{attribute 'GeneratedUsingTerminal: EJ3214-0000-0016'}
{attribute addProperty BoxType "EJ3214-0000-0016"}
{attribute addProperty Id "StatusAT %I*Status_68C33E995ValueAT %I*INT2"}
{attribute addProperty CRC "2507538081"}
{attribute addProperty Size "7"}
TYPE RTD_Inputs_Channel_9575FEA1 EXTENDS InputBase_8311D824 :
STRUCT
	{attribute addProperty Name "Status"}
	Status AT %I* : Status_68C33E99;
	{attribute addProperty Name "Value"}
	Value AT %I* : INT;
END_STRUCT
END_TYPE

(* stored: Version 1.2.0.0, ProductVersion 3.1.4024.9
   DUT RTD_Inputs_Channel_9575FEA1: Id {ce6a41fa-ecb5-4a8c-87af-b85e4a73bac5} *)
